// TIA Portal V20 export
// export: Created 2025-12-01T14:57:21.0141228Z, ExportSetting None, DisplayName Totally Integrated Automation Portal, DisplayVersion V20 Update 3, DisplayName TIA Portal Openness, DisplayVersion V20 Update 3, DisplayName TIA Portal Version Control Interface, DisplayVersion V20 Update 3, DisplayName STEP 7 Professional, DisplayVersion V20 Update 3, DisplayName STEP 7 Safety, DisplayVersion V20 Update 2, DisplayName WinCC Basic/Comfort/Advanced, DisplayVersion V20 Update 3, DisplayName WinCC Professional, DisplayVersion V20 Update 3, DisplayName WinCC Unified, DisplayVersion V20 Update 3
DATA_BLOCK "DB2120_DB_LinPot_Elev1"   // DB2120, F_DB
FAMILY : FPRI0854
VERSION : 0.0
// stored: AutoNumber false, InstanceOfName FB2132_F_LinPot_Elevador, InstanceOfType FB
"FB2132_F_LinPot_Elevador"
   // VAR_INPUT
   //    NumArmario : Int;
   //    NumLineaElev : Int;
   //    NumLineaTrans : Int;
   //    Maquina_OFF : Bool;
   //    Proteccion : Bool;
   //    Accesos : Bool;
   //    Seguridades : Bool;
   //    LimitSwitch : Bool;
   //    FEEDBACK_Elev : Bool;
   //    FEEDBACK_Trans : Bool;
   //    Rearme : Bool;
   //    Mantenimiento : Bool;
   //    QBAD_FIO_Elev : Bool;
   //    QBAD_FIO_Trans : Bool;
   //    FDB_TIME : Time;
   // END_VAR
   // VAR_OUTPUT
   //    Q_Elev : Bool;
   //    Q_Trans : Bool;
   //    ERROR_Elev : Bool;
   //    ERROR_Trans : Bool;
   //    H : Bool;
   // END_VAR
   // VAR
   //    F_FDBACK_Elev { S7_SetPoint := 'True'} : FDBACK;
   //    F_ESTOP1_Elev { S7_SetPoint := 'True'} : ESTOP1;
   //    F_FDBACK_Trans { S7_SetPoint := 'True'} : FDBACK;
   //    F_ESTOP1_Trans { S7_SetPoint := 'True'} : ESTOP1;
   // END_VAR
BEGIN
END_DATA_BLOCK
